// TIA Portal V20 export
FUNCTION_BLOCK "Pallets_Transport_System"   // FB9, LAD
{ S7_Optimized_Access := 'TRUE' }
// stored: MemoryReserve 100, SetENOAutomatically false
   VAR
      NumberOfPallet { S7_SetPoint := 'True'} : Int;
      Map : Array[1..4, 1..12] of Bool;
      MoveDirection : Int;   // 1-L, 2-Up, 3-R, 4-Down
      FoundSelectedPallet : Bool;
      CanMove : Bool;
      Station_Next_Position : Array[1..2] of Int;
      SelectedPalletFound : Bool;
   END_VAR
   VAR_TEMP
      i : Int;
      j : Int;
      k : Int;
   END_VAR
BEGIN

REGION Network 1 (SCL)
   // Sprawdzenie, które elementy sa wybrane i nadanie im nowej pozycji
   #SelectedPalletFound := FALSE;

   FOR #k := 1 TO 24 DO
       IF "Pallets_Stations".Pallets[#k].IsSelected THEN
           #SelectedPalletFound := TRUE;
           EXIT;
       END_IF;
   END_FOR;

   IF #SelectedPalletFound THEN
       #Station_Next_Position := "Pallets_Stations".Pallets[#k].Station_Current_Position;

               CASE #MoveDirection OF
                   1:
                       IF #Station_Next_Position[2] > 1 THEN  // Check Left
                           #Station_Next_Position[2] := #Station_Next_Position[2] - 1;
                       ELSE
                           #CanMove := FALSE;
                       END_IF;
                   3:
                       IF (#Station_Next_Position[2] < 12) AND // Check Right
                           ((#Station_Next_Position[1] = 2 AND #Station_Next_Position[2] < 12) OR (#Station_Next_Position[1] <> 2 AND #Station_Next_Position[2] < 11)) THEN
                           #Station_Next_Position[2] := #Station_Next_Position[2] + 1;
                       ELSE
                           #CanMove := FALSE; 
                       END_IF;
                   2:
                       IF (#Station_Next_Position[2] = 1) OR
                           ((#Station_Next_Position[1] = 1 AND #Station_Next_Position[2] = 11) OR
                           (#Station_Next_Position[1] = 2 AND #Station_Next_Position[2] = 12) OR
                           (#Station_Next_Position[1] = 3 AND #Station_Next_Position[2] = 11) OR
                           (#Station_Next_Position[1] = 4 AND #Station_Next_Position[2] = 11)) THEN
                           IF #Station_Next_Position[1] > 1 THEN
                               // Ruch w ostatniej kolumnie
                               IF #Station_Next_Position[1] = 2 AND #Station_Next_Position[2] = 12 THEN
                                   #Station_Next_Position[1] := 1;
                                   #Station_Next_Position[2] := 11;
                               ELSE
                                   #Station_Next_Position[1] := #Station_Next_Position[1] - 1;
                               END_IF;
                           ELSE
                               #CanMove := FALSE;
                           END_IF;
                       ELSE
                           #CanMove := FALSE;
                       END_IF;
                   4:
                       IF (#Station_Next_Position[2] = 1) OR
                           ((#Station_Next_Position[1] = 1 AND #Station_Next_Position[2] = 11) OR
                           (#Station_Next_Position[1] = 2 AND #Station_Next_Position[2] = 12) OR
                           (#Station_Next_Position[1] = 3 AND #Station_Next_Position[2] = 11) OR
                           (#Station_Next_Position[1] = 4 AND #Station_Next_Position[2] = 11)) THEN
                           IF #Station_Next_Position[1] < 4 THEN
                               // Ruch w ostatniej kolumnie
                               IF #Station_Next_Position[1] = 1 AND #Station_Next_Position[2] = 11 THEN
                                   #Station_Next_Position[1] := 2;
                                   #Station_Next_Position[2] := 12;
                               ELSE
                                   #Station_Next_Position[1] := #Station_Next_Position[1] + 1;
                               END_IF;
                           ELSE
                               #CanMove := FALSE;
                           END_IF;
                       ELSE
                           #CanMove := FALSE;
                       END_IF;
               END_CASE;

               "Pallets_Stations".Pallets[#k].Station_Current_Position := #Station_Next_Position;

           ELSE
               #CanMove := FALSE; // żaden pallet nie był wybrany
           END_IF;
END_REGION
END_FUNCTION_BLOCK
